FUNCTION_BLOCK FB_UML_SC_Lamp
VAR_INPUT
	bPower				: BOOL;
END_VAR
VAR_OUTPUT
	ObLamp		AT%Q*	: BOOL;
END_VAR
VAR
	nCounterOn			: INT;
	nCounterOff			: INT;
END_VAR

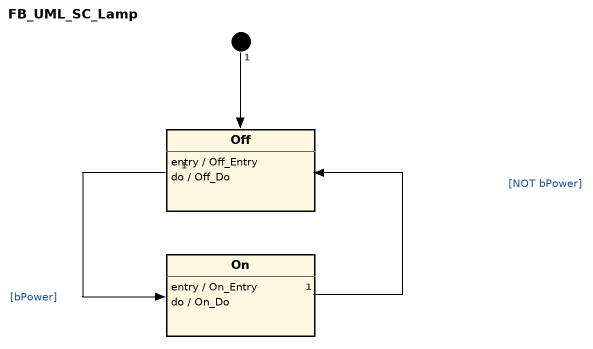
STATECHART FB_UML_SC_Lamp  // abortable
    START StartState1
    STATE Off
        entry / Off_Entry
        do / Off_Do
    STATE On
        entry / On_Entry
        do / On_Do
    StartState1 -> Off  // priority 1, on completion
    Off -> On [bPower] // priority 1, rising edge
    On -> Off [NOT bPower] // priority 1
END_STATECHART

ACTION Off_Do:
nCounterOff := nCounterOff + 1;
END_ACTION

ACTION Off_Entry:
ObLamp := FALSE;
END_ACTION

ACTION On_Do:
nCounterOn := nCounterOn + 1;
END_ACTION

ACTION On_Entry:
ObLamp := TRUE;
END_ACTION

END_FUNCTION_BLOCK

(* stored: Version 1.1.0.1, ProductVersion 3.1.4024.11
   POU FB_UML_SC_Lamp: Id {a6355891-2500-4fbe-bdcb-61b982007577}, SpecialFunc None
   Action Off_Do: Id {42f76986-0f55-4ec5-86ed-c5eb4056252a}
   Action Off_Entry: Id {c981df5c-614b-4de2-ac34-052dd1703afc}
   Action On_Do: Id {461a4f60-87b2-42a9-89f0-24a9c0cd5e66}
   Action On_Entry: Id {a59d4539-dd57-4f68-ad7a-38af7b98f61f} *)
